// TwinCAT 3 PLC project Untitled1
// ProgramVersion: 3.1.4024.0
// libraries:
//   Tc2_Standard, * (Beckhoff Automation GmbH)
//   Tc2_System, * (Beckhoff Automation GmbH)
//   Tc3_Module, * (Beckhoff Automation GmbH)
// project tree:
//   DUTs/ FlexChain.TcDUT (not stored), E_LightStates.TcDUT, E_SwitchType.TcDUT
//   GVLs/ GVL_IO.TcGVL
//   PISA/ CircuitBreakerStatus.TcTLEO, FB_PISA_Comms.TcPOU, PISA_Comms.TcDUT
//   / PlcTask.TcTTO (not stored)
//   POUs/ fbDigitalInput.TcPOU, DigitalIO.TcPOU (not stored), fbDigitalOutput.TcPOU (not stored), MAIN.TcPOU
// real-time tasks:
//   TASK PlcTask: cycle T#10ms, priority 20, ADS port 350
// I/O:
//   DEVICE Device 1 (EtherCAT), AmsNetId 5.97.60.218.2.1
//     Term 7 (EK1200)
//     Box 12 (Flexi Gateway GETC1)
//     Box 13 (EP6228-0022)
// variable links:
//   Untitled1/Untitled1 Instance <-> Device 1 (EtherCAT)/Box 13 (EP6228-0022)
//     PlcTask Inputs/GVL_IO.Encoder_Counts <-> Module 3 (IO-Link Slave)/IO-Link Port1/Counter
//     PlcTask Inputs/GVL_IO.flexChain.pdo[0] <-> Module 4 (IO-Link Slave)/IO-Link Port2_in/Process Data In
//     PlcTask Inputs/GVL_IO.flexChain.pdo[{1..12}] <-> Module 4 (IO-Link Slave)/IO-Link Port2_in/Process Data In_{1..12}  (12 links)
//   Untitled1/Untitled1 Instance <-> Device 1 (EtherCAT)/Term 7 (EK1200)/Term 10 (EL2008)
//     PlcTask Outputs/MAIN.myPisa.PisaIO.bTX <-> Channel 3/Output
//   Untitled1/Untitled1 Instance <-> Device 1 (EtherCAT)/Term 7 (EK1200)/Term 9 (EL1008)
//     PlcTask Inputs/MAIN.myPisa.PisaIO.bRX <-> Channel 3/Input

// ---- DUTs/E_LightStates.TcDUT
{attribute 'qualified_only'}
{attribute 'strict'}
TYPE E_LightStates :
(
	FAST_BLINK := 0,//set fast blink as default to indicate plc running and IO mapped at a glance. 
	ON := 1,
	SLOW_BLINK := 2,
	OFF := 3,
	
	
	COUNT  //Max value. Insert new values before to keep this as the max. Used to get max enum size when useful as an input to other function blocks.  
);
END_TYPE

// ---- DUTs/E_SwitchType.TcDUT
{attribute 'qualified_only'}
{attribute 'strict'}
TYPE E_SwitchType :
(
	NO := 0,
	NC := 1,
	COUNT :=3 //Max value. Insert new values before and update max. 
);
END_TYPE

// ---- PISA/CircuitBreakerStatus.TcTLEO
{attribute 'qualified_only'}
{attribute 'strict'}
TYPE CircuitBreakerStatus :
(
	OFF := 0,        // Device has been set OFF either manually or programatically
	ON := 1,		 // Device is ON and funcioning normally
	TRIPPED := 2,	 // An overcurrent event has tripped the device
	RESET := 3		 // A reset signal has been sent to the device but it hasn't responded yet
);
END_TYPE

// ---- PISA/PISA_Comms.TcDUT
TYPE PISA_Comms :
STRUCT
	sProductName  :STRING;
	bRX AT %I* : BIT;//INPUTS (STATUS -3.4)
	bTX AT %Q* : BIT;//OUTPUTS (CTRL +3.1)
END_STRUCT
END_TYPE

// ---- GVLs/GVL_IO.TcGVL
{attribute 'qualified_only'}

VAR_GLOBAL CONSTANT
    lightBarPDOstartIndex     : INT := 5;
    lightBarPDOsecondIndex : INT := lightBarPDOstartIndex+1;
END_VAR
VAR_GLOBAL
		Encoder_Counts AT %I* : UINT;
		
		byteArray AT %I* : ARRAY[1..8] OF BOOL;
		byteInt AT %I* : BYTE;
		flexChain : FlexChain;
		(*
		aLightCurtain AT %I* : ARRAY[1..10] OF POINTER TO BOOL := [flexChain.pdo[lightBarPDOstartIndex].0, 
																   flexChain.pdo[lightBarPDOstartIndex].1,
																   flexChain.pdo[lightBarPDOstartIndex].2,
																   flexChain.pdo[lightBarPDOstartIndex].3,
																   flexChain.pdo[lightBarPDOstartIndex].4,
																   flexChain.pdo[lightBarPDOstartIndex].5,
																   flexChain.pdo[lightBarPDOstartIndex].6,
																   flexChain.pdo[lightBarPDOstartIndex].7,
																   flexChain.pdo[lightBarPDOsecondIndex].0,
																   flexChain.pdo[lightBarPDOsecondIndex].1];
																   
																   *)
																   
																   
	aInputs AT %I* : ARRAY[1..8] OF BOOL;
	aOutputs AT %Q* : ARRAY[1..8] OF BOOL;
															   	

END_VAR

// ---- PISA/FB_PISA_Comms.TcPOU
FUNCTION_BLOCK FB_PISA_Comms
VAR_INPUT
	//bStart	: BOOL;
	//bReset	: BOOL;
	//biDirectional	: BOOL;
END_VAR
VAR CONSTANT
    cMaxChannels : INT := 16;
	cStandardChannels : INT :=4;
END_VAR

VAR
	PisaIO : PISA_Comms;
	
	bStart : BOOL := TRUE;
	biDirectional : BOOL := FALSE;
	//fbTcMessage     : FB_TcMessage ; // Function block instance for sending messages
	myDevice : POINTER TO PISA_Comms;
	
	nNumberOfDeviceChannels : UINT :=4; //Currently all PISA-M devices have 4 channels but this might change with new product releases
	//nTimerTx	: UINT;
	//nTimerRx	: UINT;
	bStartBit : BOOL;
	tStartTimeDuration	: TIME ;
	nChannelNumber	: USINT := 0 ;
	//maxNumberOfChannels UINT := 16;
	aStatus : ARRAY[1..cMaxChannels] OF CircuitBreakerStatus;
	//aChannelTripped	: ARRAY[1..nNumberOfDeviceChannels] OF BOOL;
	//aChannelOff		: ARRAY[1..nNumberOfDeviceChannels] OF BOOL;
	tpStatus	: TP	:= (PT:=T#100MS);	//Channel Status Timer
	tpGap		: TP	:= (PT:=T#100MS);	//Gap Between Channels Timer
	tpMeasure   : TP    := (PT:=T#100MS);
	cCycleTime : TIME := T#10MS;
	timeDiv : TIME := T#100MS-cCycleTime;
	rxSequenceDuration :TIME :=T#1100MS;
	minTimeToRegister :TIME :=T#5MS;
	offTime :TIME :=T#50MS;
	timer :TON;
	bReadingStatus : BOOL;
	maxPulseDuration :TIME :=T#200MS;
	shortStartPulseDuration : TIME := T#150MS;
	longStartPulseDuration : TIME := T#200MS;
	
	mostRecientTime : TIME;
	
	measuredTime : TIME ;
	
	tempStatus : CircuitBreakerStatus;
	
	//minimumTimeToTrig :TIME := T#50MS;
	
	fallingEdge: F_TRIG;
	risingEdge: R_TRIG;
	rxStartTimer: TON;
	rxSequenceTimer :TP;
	//rtRxStart	: R_Trig;
	//sigStatus: INT;
	//circuitStatus: INT;
	//E_ECB_Status: INT;
	//OFF: INT;
	//Tripped: INT;
	//ON: INT;
	
	
	nTimerRx: INT;
END_VAR

IF bStart THEN

	IF biDirectional THEN
		tStartTimeDuration	:= shortStartPulseDuration;
	ELSE
		tStartTimeDuration	:= longStartPulseDuration;
	END_IF
	
	
	timer(IN := PisaIO.bRX , PT:=tStartTimeDuration);
	fallingEdge(CLK := PisaIO.bRX);
	
	IF( PisaIO.bRX = TRUE AND NOT fallingEdge.Q AND NOT timer.Q) THEN // IF the input is high, update the running counter of the pulse duration
		mostRecientTime := timer.ET;	
	END_IF
	
	IF (fallingEdge.Q)THEN //A pulse just completed
		IF mostRecientTime >= shortStartPulseDuration - cCycleTime THEN
			bStartBit 	:= NOT bStartBit; // Will only read every other start bit but simplifies some logice and time syncing
		END_IF
	
	
	END_IF
	
	
	//rxSequenceDuration := tStartTimeDuration + 2 * timeDiv * nNumberOfDeviceChannels;
	
	//rxStartTimer(IN := PisaIO.bRX, PT := tStartTimeDuration); //Timer to detect Start BIT
	
	//IF rxStartTimer.Q THEN // The START bit was found. 
	//	bStartBit 	:= TRUE;
		//nTimerRx 	:= 0;
		
	//	tpStatus(in:=TRUE);
	//END_IF
	//rxSequenceTimer(IN := bStartBit, PT := rxSequenceDuration-tStartTimeDuration); //Timer to detect Start BIT
	
	//rxSequenceTimer.ET>
	
	(*
	timer(IN := NOT timer.Q AND bStartBit, PT := timeDiv);
	IF timer.Q THEN 
		bReadingStatus := NOT bReadingStatus; 
	END_IF
	*)
	
	///fallingEdge(CLK := bReadingStatus OR PisaIO.bRX);//Only when we transition to the next gap sig pair
	
	IF bStartBit THEN
		
	(*
		IF bReadingStatus THEN// IN STATUS (Measure the duration of the pulse in the status section of the sequence
			tpMeasure(IN:= TPStatus.Q AND PisaIO.bRX);
			measuredTime:=tpMeasure.ET;
		ELSE IF nChannelNumber > 0 THEN //IN GAP (Determine the meaning of the last pulse based on length and dave it)
			IF measuredTime > minTimeToRegister AND measuredTime <= offTime + minTimeToRegister THEN
				aStatus[nChannelNumber]	:= CircuitBreakerStatus.OFF;
			ELSIF measuredTime > offTime THEN
				aStatus[nChannelNumber]	:= CircuitBreakerStatus.Tripped;
			ELSE
				aStatus[nChannelNumber]	:= CircuitBreakerStatus.ON;
			END_IF	
		END_IF	
		
		IF fallingEdge.Q THEN
			nChannelNumber := nChannelNumber + 1;
		END_IF
		END_IF 
		*)
		IF nChannelNumber > cStandardChannels THEN //End of Sequence
			bStartBit := FALSE;
			nChannelNumber :=0;
			bReadingStatus := FALSE;
		END_IF
	END_IF
END_IF

METHOD FB_init : BOOL
VAR_INPUT
	bInitRetains : BOOL; // if TRUE, the retain variables are initialized (warm start / cold start)
	bInCopyCode : BOOL;  // if TRUE, the instance afterwards gets moved into the copy code (online change)
	sProductName : STRING;
END_VAR

VAR
	cChar: STRING;
	iDigit: UINT;
	iIndex: INT;
	sMyString: INT;
	iMyInteger: INT;
	exc : __SYSTEM.ExceptionCode;

END_VAR
PisaIO.sProductName := sProductName;
__TRY
nNumberOfDeviceChannels := STRING_TO_UINT(MID(sProductName,1,4));
__CATCH(exc)
	//TODO Throw exception with indication of unexpected character in 4th digit of product name
__ENDTRY

//PISA-M-404
//PISA-M-%i0%j
//Pisa modules follow the following naming convention where %i is the number of channels and %j is the amperage

nNumberOfDeviceChannels := iDigit;
END_METHOD

METHOD GetStatus : CircuitBreakerStatus
VAR_INPUT
	nChannel : UINT;
END_VAR
IF nChannel > 0 AND nChannel <= nNumberOfDeviceChannels THEN
	GetStatus := aStatus[nChannel];
ELSE
	//todo error
END_IF
END_METHOD

METHOD SetStatus
VAR_INPUT
	nChannel : UINT;
	sStatus : CircuitBreakerStatus;
END_VAR
IF(sStatus = CircuitBreakerStatus.ON OR sStatus = CircuitBreakerStatus.RESET) THEN
	aStatus[nChannel] := CircuitBreakerStatus.RESET;
END_IF

//TODO logic to transmit reset signals or off signal
END_METHOD

END_FUNCTION_BLOCK

// ---- POUs/fbDigitalInput.TcPOU
FUNCTION_BLOCK fbDigitalInput EXTENDS DigitalIO

END_FUNCTION_BLOCK

// ---- POUs/MAIN.TcPOU
PROGRAM MAIN

VAR
	
	
	bGreenBtn    : POINTER TO BOOL:= ADR(GVL_IO.aInputs[1]);
	bRedBtn		: POINTER TO BOOL:= ADR(GVL_IO.aInputs[2]);
	bLight : POINTER TO BOOL := ADR(GVL_IO.aOutputs[1]);

	fbStartInput : fbDigitalInput(ioBitRef := ADR(GVL_IO.aInputs[1]), switchType := E_SwitchType.NO);
	fbStopInput : fbDigitalInput(ioBitRef := ADR(GVL_IO.aInputs[2]), switchType := E_SwitchType.NC);
	fbLightOutput : fbDigitalOutput(ioBitRef := ADR(GVL_IO.aOutputs[1]), switchType := E_SwitchType.NO);
	light2 : fbDigitalOutput(ioBitRef := ADR(GVL_IO.aOutputs[2]), switchType := E_SwitchType.NO);
	CurrentState: UINT  := TO_UINT(E_LightStates.FAST_BLINK);
	
	fbCounter : CTU;

	timedLight : BOOL;
	timer :TON;

	aLightCurtain : ARRAY[1..10] OF BOOL; 
	
	myPisa : FB_PISA_Comms(sProductName := 'PISA-M-4CL2');
	
	cbStates : ARRAY[1..4] OF CircuitBreakerStatus;
	i: INT;
END_VAR




GVL_IO.aOutputs[8] := GVL_IO.aInputs[8]; // Output 8 mirrors input 8


IF fbStartInput.Get() THEN
		fbLightOutput.Set(TRUE);
ELSE 
		fbLightOutput.Set(FALSE);
END_IF

//bGreenBtn := aInputs[1];


(*
IF bGreenBtn^ THEN
		bLight^:=TRUE;
ELSE 
		bLight^:=FALSE;
END_IF
*)
myPisa();

FOR i := 1 TO 4 DO
    cbStates[i] := myPisa.GetStatus(i);
END_FOR;

fbCounter(CU:=fbStartInput.Get(),CU:=fbStartInput.Get(), RESET :=fbStopInput.Get() ,PV := UINT_TO_WORD(E_LightStates.COUNT));
CurrentState:=fbCounter.CV;


	aLightCurtain[1]:= (GVL_IO.flexChain.pdo[GVL_IO.lightBarPDOstartIndex] AND 2#0000_0000_0000_0001) <> 0;
	aLightCurtain[2]:= (GVL_IO.flexChain.pdo[GVL_IO.lightBarPDOstartIndex] AND 2#0000_0000_0000_0010) <> 0;
	aLightCurtain[3]:= (GVL_IO.flexChain.pdo[GVL_IO.lightBarPDOstartIndex] AND 2#0000_0000_0000_0100) <> 0;
	aLightCurtain[4]:= (GVL_IO.flexChain.pdo[GVL_IO.lightBarPDOstartIndex] AND 2#0000_0000_0000_1000) <> 0;
	aLightCurtain[5]:= (GVL_IO.flexChain.pdo[GVL_IO.lightBarPDOstartIndex] AND 2#0000_0000_0001_0000) <> 0;
	aLightCurtain[6]:= (GVL_IO.flexChain.pdo[GVL_IO.lightBarPDOstartIndex] AND 2#0000_0000_0010_0000) <> 0;
	aLightCurtain[7]:= (GVL_IO.flexChain.pdo[GVL_IO.lightBarPDOstartIndex] AND 2#0000_0000_0100_0000) <> 0;
	aLightCurtain[8]:= (GVL_IO.flexChain.pdo[GVL_IO.lightBarPDOstartIndex] AND 2#0000_0000_1000_0000) <> 0;
	aLightCurtain[9]:= (GVL_IO.flexChain.pdo[GVL_IO.lightBarPDOsecondIndex] AND 2#0000_0000_0000_0001) <> 0;
	aLightCurtain[10]:= (GVL_IO.flexChain.pdo[GVL_IO.lightBarPDOsecondIndex] AND 2#0000_0000_0000_0010) <> 0;
								


CASE CurrentState OF
    E_LightStates.OFF:
		fbLightOutput.Set(FALSE);
    E_LightStates.ON:
		fbLightOutput.Set(TRUE);
    E_LightStates.SLOW_BLINK:
		timer(IN := NOT timer.Q, PT := T#1S500MS);
		IF timer.Q THEN 
			timedLight := NOT timedLight; 
		END_IF
		fbLightOutput.Set(timedLight);
    E_LightStates.FAST_BLINK:
		timer(IN := NOT timer.Q, PT := T#0S500MS);
		IF timer.Q THEN 
			timedLight := NOT timedLight; 
		END_IF
		fbLightOutput.Set(timedLight);
ELSE
		fbLightOutput.Set(FALSE);
		fbCounter(RESET:=TRUE);
		
END_CASE

IF GVL_IO.Encoder_Counts > 500 THEN
	light2.Set(TRUE);
ELSE
	light2.Set(FALSE);		

END_IF

END_PROGRAM
